// TwinCAT 3 PLC project Untitled1
// ProgramVersion: 3.1.4023.0
// libraries:
//   Tc2_Standard, * (Beckhoff Automation GmbH)
//   Tc2_System, * (Beckhoff Automation GmbH)
//   Tc2_Utilities, * (Beckhoff Automation GmbH)
//   Tc3_Module, * (Beckhoff Automation GmbH)
// project tree:
//   DUTs/ Measurement_Event.TcDUT
//   GVLs/ GVL.TcGVL
//   / PlcTask.TcTTO
//   POUs/ FB_CheckOperation.TcPOU, FB_MeasurementStarted.TcPOU, MAIN.TcPOU, MeasurementBuffer.TcPOU
// real-time tasks:
//   TASK PlcTask: cycle T#10ms, priority 20, ADS port 350

CONFIGURATION Untitled1
    RESOURCE PLC ON TwinCAT3
        TASK PlcTask(INTERVAL := T#10ms, PRIORITY := 20);
        PROGRAM MAIN WITH PlcTask : MAIN;
    END_RESOURCE
END_CONFIGURATION

// ---- DUTs/Measurement_Event.TcDUT
TYPE Measurement_Event :
STRUCT
	
END_STRUCT
END_TYPE

// ---- GVLs/GVL.TcGVL
{attribute 'qualified_only'}
VAR_GLOBAL
	OperationStart AT %I* : BOOL  ;
	OperationStop AT %I* : BOOL ;
	OperationNext AT %I* : BOOL ;
 
	LoadMeasurementStart AT %Q* : BOOL;
	LoadMeasurementWait AT %Q* : BOOL;
	LoadMeasurementStop AT %Q* : BOOL; 
	 
END_VAR		

VAR_GLOBAL CONSTANT
	MAX_BUFFER_SIZE : UDINT := 1000	;
	HighestForceValueBufferSize : INT := 10; 
END_VAR

// ---- POUs/MAIN.TcPOU
PROGRAM MAIN
VAR
	fbCheckOperation : FB_CheckOperation;
	
END_VAR

// CHECK
fbCheckOperation();

END_PROGRAM

// ---- POUs/FB_CheckOperation.TcPOU
FUNCTION_BLOCK FB_CheckOperation
VAR
	
	StartTimer : TON;
	TimerDone : BOOL;
	
	Counter : CTU; 
	ResetCommand : BOOL; 
END_VAR

StartTimer(IN:= GVL.OperationStart , PT:= T#2S);
TimerDone := StartTimer.Q; 

IF TimerDone THEN  
	gvl.LoadMeasurementStart := TRUE;
ELSE
	gvl.LoadMeasurementWait := TRUE;
END_IF

//Counter(
	//CU:=TimerDone , 
	//RESET:= ResetCommand , 
	//PV:= 5);

END_FUNCTION_BLOCK

// ---- POUs/FB_MeasurementStarted.TcPOU
FUNCTION_BLOCK FB_MeasurementStarted
VAR
	
	MeasurementValuesBuffer : ARRAY[1..gvl.MaxLoadMeasurementBufferSize] OF BYTE; 
	CurrentBufferIndiex : INT := 0;
	fbBuffer : FB_MemRingBuffer; 
	
	bReset : BOOL := TRUE; 
	bAdd : BOOL := TRUE;
	bGet : BOOL := TRUE;
	bRemove : BOOL := TRUE;
END_VAR

END_FUNCTION_BLOCK

// ---- POUs/MeasurementBuffer.TcPOU
FUNCTION_BLOCK MeasurementBuffer
VAR
	MemRingBuffer : FB_MemRingBuffer;
	BufferArray : ARRAY[0..GVL.MAX_BUFFER_SIZE] OF BYTE;
	
END_VAR

METHOD AddMeasurement
VAR_INPUT
END_VAR
END_METHOD

END_FUNCTION_BLOCK
